PROGRAM MAIN
VAR
END_VAR

F_ConsumeTime(50);

END_PROGRAM

(* stored: Version 1.1.0.1, ProductVersion 3.1.4026.18
   POU MAIN: Id {dcb5153a-8e56-4028-9de5-b12ccc551da6}, SpecialFunc None *)
